{attribute 'OPC.UA.DA.StructuredType' := '1'}
TYPE ST_VentilationSetParameters :
STRUCT
	bHeatingModeAlgorithm : BOOL;
	bHeatingModeManual : BOOL;
END_STRUCT
END_TYPE

(* stored: Version 1.1.0.1, ProductVersion 3.1.4024.10
   DUT ST_VentilationSetParameters: Id {c790bc73-ec9a-40f9-9e95-392c8b3f7262} *)
